FUNCTION_BLOCK Counter
VAR_INPUT
	Step: BOOL;
	Smer: BOOL;
	Stikalo: BOOL;
END_VAR
VAR_OUTPUT
	poz: WORD;
END_VAR
VAR
	R_TRIG_0: R_TRIG;
	CTUD_0: Tc2_Standard.CTUD;
	R_TRIG_1: Tc2_Standard.R_TRIG;
END_VAR

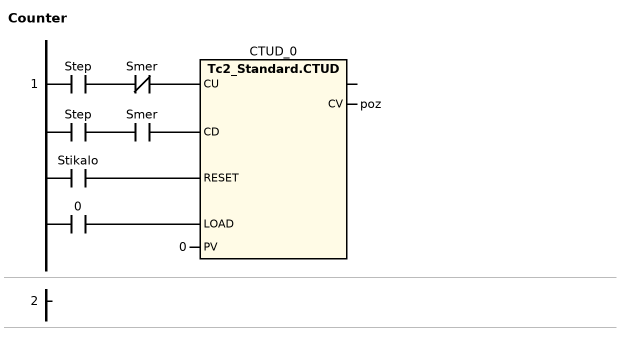
// NETWORK 1
CTUD_0(CU := Step AND NOT Smer, CD := Step AND Smer, RESET := Stikalo, LOAD := 0, PV := 0, CV => poz); // Tc2_Standard.CTUD

// NETWORK 2

END_FUNCTION_BLOCK

(* stored: Version 1.1.0.1, ProductVersion 3.1.4024.12
   POU Counter: Id {5966a17f-a092-4f19-9896-7a9d2d0bf9b9}, SpecialFunc None *)
